// TIA Portal V19 export
FUNCTION "Speed Control" : Void   // FC1, LAD
{ S7_Optimized_Access := 'TRUE' }
// stored: SetENOAutomatically false
   VAR_TEMP   // added for the SCL form of the ladder/FBD networks
      _w1 : Bool;
      _w2 : Bool;
   END_VAR
BEGIN

REGION Network 1: KP8 bit that is toggled each time is pressed
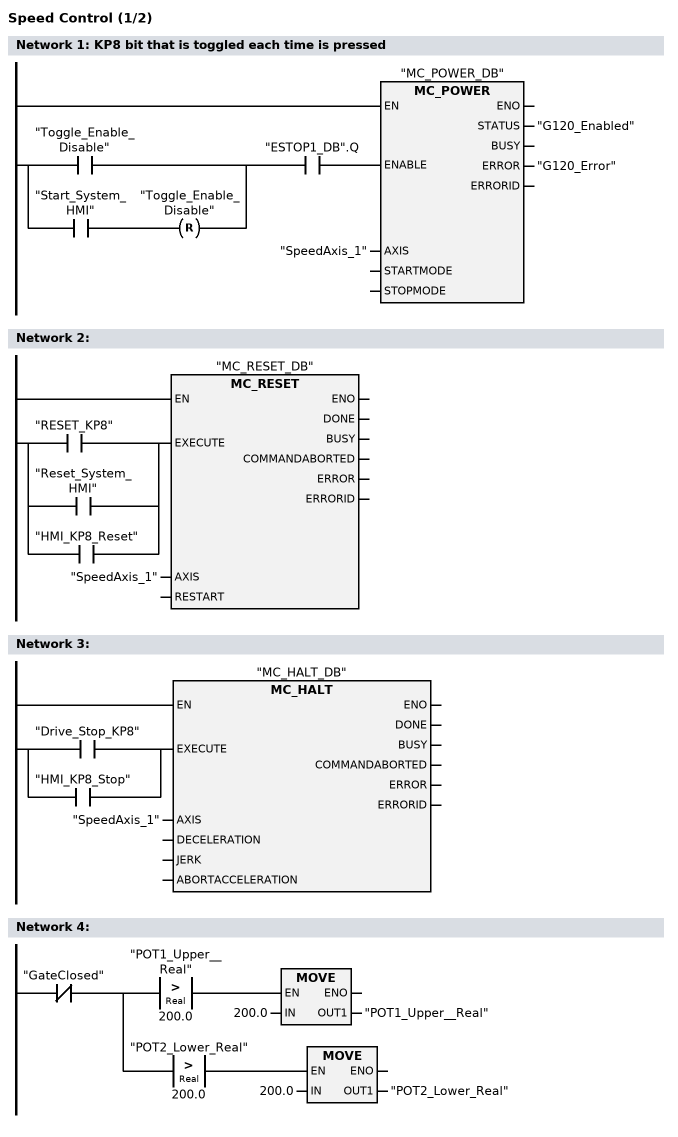
   RUNG wire#powerrail
      "MC_POWER_DB".MC_POWER(Enable := wire#w2, Axis := "SpeedAxis_1", StartMode :=, StopMode :=, Status => "G120_Enabled", Busy =>, Error => "G120_Error", ErrorId =>)
   END_RUNG
   RUNG wire#powerrail
      Contact( "Toggle_Enable_Disable" )
      wire#w1
      Contact( "ESTOP1_DB".Q )
   END_RUNG wire#w2
   RUNG wire#powerrail
      Contact( "Start_System_HMI" )
      R_Coil( "Toggle_Enable_Disable" )
   END_RUNG wire#w1
   // the same network as SCL:
   #_w1 := "Toggle_Enable_Disable";
   IF "Start_System_HMI" THEN "Toggle_Enable_Disable" := FALSE; END_IF;
   "MC_POWER_DB"(Enable := (#_w1 OR "Start_System_HMI") AND "ESTOP1_DB".Q,   // MC_POWER
                 Axis := "SpeedAxis_1",
                 Status => "G120_Enabled",
                 Error => "G120_Error");
END_REGION

REGION Network 2
   RUNG wire#powerrail
      "MC_RESET_DB".MC_RESET(Execute := wire#w1, Axis := "SpeedAxis_1", Restart :=, Done =>, Busy =>, CommandAborted =>, Error =>, ErrorId =>)
   END_RUNG
   RUNG wire#powerrail
      Contact( "RESET_KP8" )
   END_RUNG wire#w1
   RUNG wire#powerrail
      Contact( "Reset_System_HMI" )
   END_RUNG wire#w1
   RUNG wire#powerrail
      Contact( "HMI_KP8_Reset" )
   END_RUNG wire#w1
   // the same network as SCL:
   "MC_RESET_DB"(Execute := "RESET_KP8" OR "Reset_System_HMI" OR "HMI_KP8_Reset", Axis := "SpeedAxis_1");   // MC_RESET
END_REGION

REGION Network 3
   RUNG wire#powerrail
      "MC_HALT_DB".MC_HALT(Execute := wire#w1, Axis := "SpeedAxis_1", Deceleration :=, Jerk :=, AbortAcceleration :=, Done =>, Busy =>, CommandAborted =>, Error =>, ErrorId =>)
   END_RUNG
   RUNG wire#powerrail
      Contact( "Drive_Stop_KP8" )
   END_RUNG wire#w1
   RUNG wire#powerrail
      Contact( "HMI_KP8_Stop" )
   END_RUNG wire#w1
   // the same network as SCL:
   "MC_HALT_DB"(Execute := "Drive_Stop_KP8" OR "HMI_KP8_Stop", Axis := "SpeedAxis_1");   // MC_HALT
END_REGION

REGION Network 4
   RUNG wire#powerrail
      I_Contact( "GateClosed" )
      wire#w1
      { S7_Templates := "SrcType := Real" } GT_Contact(in1 := "POT1_Upper__Real", in2 := 200.0)
      Move(in := 200.0, out1 => "POT1_Upper__Real")
   END_RUNG
   RUNG wire#w1
      { S7_Templates := "SrcType := Real" } GT_Contact(in1 := "POT2_Lower_Real", in2 := 200.0)
      Move(in := 200.0, out1 => "POT2_Lower_Real")
   END_RUNG
   // the same network as SCL:
   IF NOT "GateClosed" AND ("POT1_Upper__Real" > 200.0) THEN "POT1_Upper__Real" := 200.0; END_IF;
   IF NOT "GateClosed" AND ("POT2_Lower_Real" > 200.0) THEN "POT2_Lower_Real" := 200.0; END_IF;
END_REGION

REGION Network 5
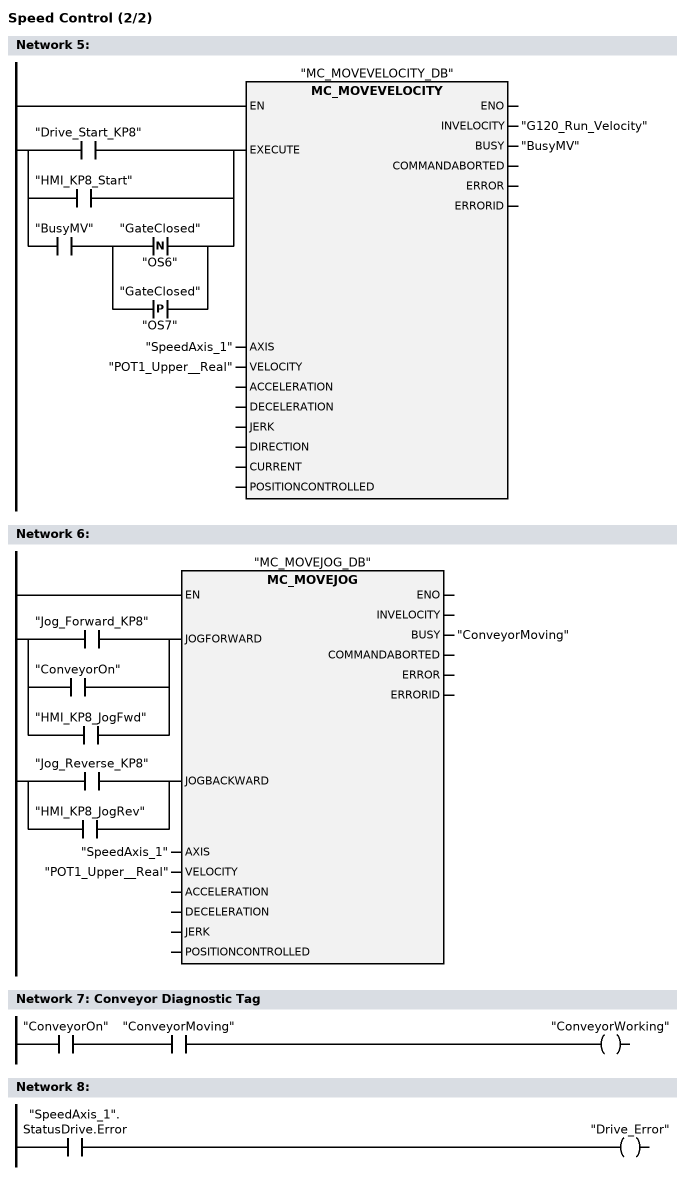
   RUNG wire#powerrail
      "MC_MOVEVELOCITY_DB".MC_MOVEVELOCITY(Execute := wire#w2, Axis := "SpeedAxis_1", Velocity := "POT1_Upper__Real", Acceleration :=, Deceleration :=, Jerk :=, Direction :=, Current :=, PositionControlled :=, InVelocity => "G120_Run_Velocity", Busy => "BusyMV", CommandAborted =>, Error =>, ErrorId =>)
   END_RUNG
   RUNG wire#powerrail
      Contact( "Drive_Start_KP8" )
   END_RUNG wire#w2
   RUNG wire#powerrail
      Contact( "HMI_KP8_Start" )
   END_RUNG wire#w2
   RUNG wire#powerrail
      Contact( "BusyMV" )
      wire#w1
      N_Contact(operand := "GateClosed", bit := "OS6")
   END_RUNG wire#w2
   RUNG wire#w1
      P_Contact(operand := "GateClosed", bit := "OS7")
   END_RUNG wire#w2
   // the same network as SCL:
   #_w1 := "BusyMV" AND NOT "GateClosed" AND "OS6";   // falling edge of "GateClosed"
   "OS6" := "GateClosed";
   #_w2 := "BusyMV" AND "GateClosed" AND NOT "OS7";   // rising edge of "GateClosed"
   "OS7" := "GateClosed";
   "MC_MOVEVELOCITY_DB"(Execute := "Drive_Start_KP8" OR "HMI_KP8_Start" OR #_w1 OR #_w2,   // MC_MOVEVELOCITY
                        Axis := "SpeedAxis_1",
                        Velocity := "POT1_Upper__Real",
                        InVelocity => "G120_Run_Velocity",
                        Busy => "BusyMV");
END_REGION

REGION Network 6
   RUNG wire#powerrail
      "MC_MOVEJOG_DB".MC_MOVEJOG(JogForward := wire#w1, JogBackward := wire#w2, Axis := "SpeedAxis_1", Velocity := "POT1_Upper__Real", Acceleration :=, Deceleration :=, Jerk :=, PositionControlled :=, InVelocity =>, Busy => "ConveyorMoving", CommandAborted =>, Error =>, ErrorId =>)
   END_RUNG
   RUNG wire#powerrail
      Contact( "Jog_Forward_KP8" )
   END_RUNG wire#w1
   RUNG wire#powerrail
      Contact( "ConveyorOn" )
   END_RUNG wire#w1
   RUNG wire#powerrail
      Contact( "HMI_KP8_JogFwd" )
   END_RUNG wire#w1
   RUNG wire#powerrail
      Contact( "Jog_Reverse_KP8" )
   END_RUNG wire#w2
   RUNG wire#powerrail
      Contact( "HMI_KP8_JogRev" )
   END_RUNG wire#w2
   // the same network as SCL:
   "MC_MOVEJOG_DB"(JogForward := "Jog_Forward_KP8" OR "ConveyorOn" OR "HMI_KP8_JogFwd",   // MC_MOVEJOG
                   JogBackward := "Jog_Reverse_KP8" OR "HMI_KP8_JogRev",
                   Axis := "SpeedAxis_1",
                   Velocity := "POT1_Upper__Real",
                   Busy => "ConveyorMoving");
END_REGION

REGION Network 7: Conveyor Diagnostic Tag
   RUNG wire#powerrail
      Contact( "ConveyorOn" )
      Contact( "ConveyorMoving" )
      Coil( "ConveyorWorking" )
   END_RUNG
   // the same network as SCL:
   "ConveyorWorking" := "ConveyorOn" AND "ConveyorMoving";
END_REGION

REGION Network 8
   RUNG wire#powerrail
      Contact( "SpeedAxis_1".StatusDrive.Error )
      Coil( "Drive_Error" )
   END_RUNG
   // the same network as SCL:
   "Drive_Error" := "SpeedAxis_1".StatusDrive.Error;
END_REGION
END_FUNCTION
